// TIA Portal V19 export
DATA_BLOCK "ControlNodes"   // DB30
// stored: Access Published, MemoryReserve 100, Namespace Unit2.EM3
   VAR
      em { ExternalWritable := 'False'} : "LAF_typeEmControlNode";
      jobs { ExternalWritable := 'False'} : "LAF_typeJobs";
      sequence { ExternalWritable := 'False'} : "LAF_typeSequence";
      cm1SV112_Constraint1_Axis : "LBC_typeAxisSimpleControlNode_1";
      cm2SV113_Constraint2_Axis { S7_SetPoint := 'True'} : "LBC_typeAxisSimpleControlNode_1";
      cm3SV115_Screw1_Axis { S7_SetPoint := 'True'} : "LEXCHANGETRAY_typeAxisSimpleControlNode_2";
      cm4SV116_Screw2_Axis { S7_SetPoint := 'True'} : "LEXCHANGETRAY_typeAxisSimpleControlNode_2";
      cm6SlideCylinder1 { S7_SetPoint := 'True'} : "LBC_Simple_typeTwoWayActuatorControlNode";
      cm7hookClawCylinder1 { S7_SetPoint := 'True'} : "LBC_Simple_typeTwoWayActuatorControlNode";
      cm8SlideCylinder2 { S7_SetPoint := 'True'} : "LBC_Simple_typeTwoWayActuatorControlNode";
      cm9hookClawCylinder2 { S7_SetPoint := 'True'} : "LBC_Simple_typeTwoWayActuatorControlNode";
      cm10SignalTM : "LEXCHANGETRAY_typeConstraintWorkstationIoSignalControlNode";
      cm11PressureGaugeRs485 { S7_SetPoint := 'True'} : "typePressureGuageRs485ControlNode";
   END_VAR
BEGIN
   em.status.enabled := true;
   cm1SV112_Constraint1_Axis.commandConfiguration.posAbsolute.position := 50.0;
   cm1SV112_Constraint1_Axis.commandConfiguration.posAbsolute.velocity := 50.0;
END_DATA_BLOCK
